// TwinCAT 3 PLC project TSG_swash_Neusiedl
// ProgramVersion: 3.1.4023.0
// libraries:
//   EfficientIO Communicator, * (EfficientIO)
//   Lynus Energy Basic, * (Lynus AG)
//   Lynus Energy ModbusTCP, * (Lynus AG)
//   Lynus Persistent Data V1, * (Lynus AG)
//   Lynus Standards, * (Lynus AG)
//   Tc2_MBus, * (Beckhoff Automation GmbH)
//   Tc2_ModbusSrv, * (Beckhoff Automation GmbH)
//   Tc2_Standard, * (Beckhoff Automation GmbH)
//   Tc2_System, * (Beckhoff Automation GmbH)
//   Tc2_Utilities, * (Beckhoff Automation GmbH)
//   Tc3_Module, * (Beckhoff Automation GmbH)
// project tree:
//   / FastTasks.TcTTO, PlcTask.TcTTO, SlowTasks.TcTTO
//   FB/ FB_ModBus_100Registers_FC4.TcPOU, FB_ModBus_100Registers_FC3.TcPOU, F_DWORD_TO_FLOAT32.TcPOU
//   POUs/ prgComLynus.TcPOU, prgEM.TcPOU, prgModbus.TcPOU, prgPersistent.TcPOU (not stored), prgPV.TcPOU, prgRWLynus.TcPOU, prgVarLynus.TcPOU, prgWCounter.TcPOU, prgWCounter_old.TcPOU (excluded from build), prg_SystemTime.TcPOU (not stored)
// real-time tasks:
//   TASK PlcTask: cycle T#10ms, priority 20, ADS port 350
//   TASK SlowTasks: cycle T#20ms, priority 21, ADS port 351
//   TASK FastTasks: cycle T#5ms, priority 19, ADS port 352
// I/O:
//   DEVICE Device 1 (Beckhoff CCAT)
//   DEVICE Device 3 (CX-BK)
//     Box 1 (CX-BK)
// variable links:
//   TSG_swash_Neusiedl/TSG_swash_Neusiedl Instance <-> Device 3 (CX-BK)/Box 1 (CX-BK)
//     FastTasks Inputs/prgWCounter.stComIn/D <-> Term 2 (KL6781)/Channel 1/Data In 0
//     FastTasks Inputs/prgWCounter.stComIn/D @bit {8..168 step 8} <-> Term 2 (KL6781)/Channel 1/Data In {1..21}  (21 links)
//     FastTasks Inputs/prgWCounter.stComIn/Status <-> Term 2 (KL6781)/Channel 1/Status
//     FastTasks Outputs/prgWCounter.stComOut/Ctrl <-> Term 2 (KL6781)/Channel 1/Ctrl
//     FastTasks Outputs/prgWCounter.stComOut/D <-> Term 2 (KL6781)/Channel 1/Data Out 0
//     FastTasks Outputs/prgWCounter.stComOut/D @bit {8..168 step 8} <-> Term 2 (KL6781)/Channel 1/Data Out {1..21}  (21 links)
//     PlcTask Inputs/prgEM.fbEM1.fbKL3403.byStateCH1 <-> Term 3 (KL3403)/Channel 1/State
//     PlcTask Inputs/prgEM.fbEM1.fbKL3403.byStateCH2 <-> Term 3 (KL3403)/Channel 2/State
//     PlcTask Inputs/prgEM.fbEM1.fbKL3403.byStateCH3 <-> Term 3 (KL3403)/Channel 3/State
//     PlcTask Inputs/prgEM.fbEM1.fbKL3403.iDataInCH1 <-> Term 3 (KL3403)/Channel 1/Data In
//     PlcTask Inputs/prgEM.fbEM1.fbKL3403.iDataInCH2 <-> Term 3 (KL3403)/Channel 2/Data In
//     PlcTask Inputs/prgEM.fbEM1.fbKL3403.iDataInCH3 <-> Term 3 (KL3403)/Channel 3/Data In
//     PlcTask Inputs/prgEM.fbKBusState.uiKBusState_OUT <-> Inputs/State
//     PlcTask Outputs/prgEM.fbEM1.fbKL3403.byCntrCH1 <-> Term 3 (KL3403)/Channel 1/Ctrl
//     PlcTask Outputs/prgEM.fbEM1.fbKL3403.byCntrCH2 <-> Term 3 (KL3403)/Channel 2/Ctrl
//     PlcTask Outputs/prgEM.fbEM1.fbKL3403.byCntrCH3 <-> Term 3 (KL3403)/Channel 3/Ctrl

CONFIGURATION TSG_swash_Neusiedl
    RESOURCE PLC ON TwinCAT3
        TASK FastTasks(INTERVAL := T#5ms, PRIORITY := 19);
        TASK PlcTask(INTERVAL := T#10ms, PRIORITY := 20);
        TASK SlowTasks(INTERVAL := T#20ms, PRIORITY := 21);
        PROGRAM prgRWLynus WITH FastTasks : prgRWLynus;
        PROGRAM prgVarLynus WITH FastTasks : prgVarLynus;
        PROGRAM prgWCounter WITH FastTasks : prgWCounter;
        PROGRAM prgPV WITH PlcTask : prgPV;
        PROGRAM prgEM WITH PlcTask : prgEM;
        PROGRAM prgModbus WITH PlcTask : prgModbus;
        PROGRAM prgPersistent WITH PlcTask : prgPersistent;
        PROGRAM prgComLynus WITH SlowTasks : prgComLynus;
    END_RESOURCE
END_CONFIGURATION

// ---- POUs/prgRWLynus.TcPOU
PROGRAM prgRWLynus
VAR
	fbRW1		: FB_ReadWrite_V2;
END_VAR

fbRW1(eUploadType:= eSelectDataUploadType.e_Change_Intervall5min, bBusy=> , bError=> , udiErrorCodeOut=> , eErrorReadWrite_Out=> );

END_PROGRAM

// ---- POUs/prgVarLynus.TcPOU
PROGRAM prgVarLynus
VAR
	fbVar			: FB_VarInfo;
END_VAR

fbVar(
	bReadInfo:= , 
	eTMCFile:= eSelectTMCFile.eDontUseTMCFile, 
	eSavePositionTMCFile:= eSavePositionOnPLC.ePostionHardDisk, 
	udiCounterFoundVariables=> , 
	bError=> , 
	bBusy=> , 
	byProgress=> , 
	udiErrorCodeOut=> , 
	eErrorVarInfo_Out=> , 
	sVarWithError=> );

END_PROGRAM

// ---- POUs/prgWCounter.TcPOU
PROGRAM prgWCounter
VAR
	fbMBusKL6781 : FB_MBUSKL6781;
	stComIn    AT %I*	:	ST_KL6781inData22B;
	stComOut   AT %Q*	:	ST_KL6781outData22B;
	stCom				:	ST_MBUS_Communication;
	fb_Mbus_11				: 	FB_MBUS_General_Water;
	fb_Mbus_12				: 	FB_MBUS_General_Water;
	fb_Mbus_13				: 	FB_MBUS_General_Water;
	fb_Mbus_14				: 	FB_MBUS_General_Water;
	fb_Mbus_15				: 	FB_MBUS_General_Water;
	fb_Mbus_16				: 	FB_MBUS_General_Water;
	fb_Mbus_17				: 	FB_MBUS_General_Water;
	fbmbusScan	: FB_MBUS_Scan;
	m_StartScan: BOOL;
	FB_ChangeAdress : FB_MBUS_ChangeAdr;
	lr_Water_Zisterne_Entnahme					: LREAL;						//{#lynus.ag#()}
	lr_Water_Frisch_Noteinspeisung				: LREAL;						//{#lynus.ag#()}
	lr_Water_Frischwasser_SB					: LREAL;						//{#lynus.ag#()}
	lr_Water_Innenreinigung						: LREAL;						//{#lynus.ag#()}
	lr_Water_Frisch_Absperrung_PO				: LREAL;						//{#lynus.ag#()}
	lr_Water_Absperrung_Zisterne				: LREAL;						//{#lynus.ag#()}
	lr_Water_FW_Zulauf_Zisterne					: LREAL;						//{#lynus.ag#()}
			
	m_Done			: BOOL;
	
END_VAR
VAR PERSISTENT
	lr_Water_Zisterne_Entnahme_LD				: LREAL;						//{#lynus.ag#()}
	lr_Water_Frisch_Noteinspeisung_LD			: LREAL;						//{#lynus.ag#()}
	lr_Water_Frischwasser_SB_LD					: LREAL;						//{#lynus.ag#()}
	lr_Water_Innenreinigung_LD					: LREAL;						//{#lynus.ag#()}
	lr_Water_Frisch_Absperrung_PO_LD			: LREAL;						//{#lynus.ag#()}
	lr_Water_Absperrung_Zisterne_LD				: LREAL;						//{#lynus.ag#()}
	lr_Water_FW_Zulauf_Zisterne_LD				: LREAL;						//{#lynus.ag#()}
	
	lr_Water_Zisterne_Entnahme_Old			: LREAL;						
	lr_Water_Frisch_Noteinspeisung_Old		: LREAL;						
	lr_Water_Frischwasser_SB_Old			: LREAL;						
	lr_Water_Innenreinigung_Old				: LREAL;						
	lr_Water_Frisch_Absperrung_PO_Old		: LREAL;						
	lr_Water_Absperrung_Zisterne_Old		: LREAL;						
	lr_Water_FW_Zulauf_Zisterne_Old			: LREAL;	
END_VAR



	
		

	
fbMBusKL6781(
	usiRetries:= , 
	bStart:= , 
	bDisabled:= , 
	bBusy=> , 
	bReady=> , 
	bError=> , 
	eError=> , 
	stComIn:= stComIn, 
	stComOut:= stComOut, 
	stCom:= stCom);

fb_Mbus_11(
	usiAddress:= 11 , 
	stSecAdr:= , 
	eBaudrate:= E_MBUS_Baudrate.eMBus_Baud2400, 
	bStart:= TRUE, 
	bSND_NKE:= , 
	bReadInit:= , 
	tMinSendTime:= T#10S , 
	bDisabled:= , 
	bBusy=> , 
	bReady=> , 
	bError=> , 
	eError=> , 
	dwIdNumber=> , 
	byStatus=> , 
	byGEN=> , 
	byCounter=> , 
	usiRecivedAdr=> , 
	eMedium=> , 
	sMan=> , 
	stVolume=> , 
	stFlow=> , 
	stCom:= stCom);
	
fb_Mbus_12(
	usiAddress:= 12 , 
	stSecAdr:= , 
	eBaudrate:= E_MBUS_Baudrate.eMBus_Baud2400, 
	bStart:= TRUE, 
	bSND_NKE:= , 
	bReadInit:= , 
	tMinSendTime:= T#10S , 
	bDisabled:= , 
	bBusy=> , 
	bReady=> , 
	bError=> , 
	eError=> , 
	dwIdNumber=> , 
	byStatus=> , 
	byGEN=> , 
	byCounter=> , 
	usiRecivedAdr=> , 
	eMedium=> , 
	sMan=> , 
	stVolume=> , 
	stFlow=> , 
	stCom:= stCom);
	
fb_Mbus_13(
	usiAddress:= 13 , 
	stSecAdr:= , 
	eBaudrate:= E_MBUS_Baudrate.eMBus_Baud2400, 
	bStart:= TRUE, 
	bSND_NKE:= , 
	bReadInit:= , 
	tMinSendTime:= T#10S , 
	bDisabled:= , 
	bBusy=> , 
	bReady=> , 
	bError=> , 
	eError=> , 
	dwIdNumber=> , 
	byStatus=> , 
	byGEN=> , 
	byCounter=> , 
	usiRecivedAdr=> , 
	eMedium=> , 
	sMan=> , 
	stVolume=> , 
	stFlow=> , 
	stCom:= stCom);	
	
fb_Mbus_14(
	usiAddress:= 14 , 
	stSecAdr:= , 
	eBaudrate:= E_MBUS_Baudrate.eMBus_Baud2400, 
	bStart:= TRUE, 
	bSND_NKE:= , 
	bReadInit:= , 
	tMinSendTime:= T#10S , 
	bDisabled:= , 
	bBusy=> , 
	bReady=> , 
	bError=> , 
	eError=> , 
	dwIdNumber=> , 
	byStatus=> , 
	byGEN=> , 
	byCounter=> , 
	usiRecivedAdr=> , 
	eMedium=> , 
	sMan=> , 
	stVolume=> , 
	stFlow=> , 
	stCom:= stCom);
	
fb_Mbus_15(
	usiAddress:= 15 , 
	stSecAdr:= , 
	eBaudrate:= E_MBUS_Baudrate.eMBus_Baud2400, 
	bStart:= TRUE, 
	bSND_NKE:= , 
	bReadInit:= , 
	tMinSendTime:= T#10S , 
	bDisabled:= , 
	bBusy=> , 
	bReady=> , 
	bError=> , 
	eError=> , 
	dwIdNumber=> , 
	byStatus=> , 
	byGEN=> , 
	byCounter=> , 
	usiRecivedAdr=> , 
	eMedium=> , 
	sMan=> , 
	stVolume=> , 
	stFlow=> , 
	stCom:= stCom);

fb_Mbus_16(
	usiAddress:= 16 , 
	stSecAdr:= , 
	eBaudrate:= E_MBUS_Baudrate.eMBus_Baud2400, 
	bStart:= TRUE, 
	bSND_NKE:= , 
	bReadInit:= , 
	tMinSendTime:= T#10S , 
	bDisabled:= , 
	bBusy=> , 
	bReady=> , 
	bError=> , 
	eError=> , 
	dwIdNumber=> , 
	byStatus=> , 
	byGEN=> , 
	byCounter=> , 
	usiRecivedAdr=> , 
	eMedium=> , 
	sMan=> , 
	stVolume=> , 
	stFlow=> , 
	stCom:= stCom);

fb_Mbus_17(
	usiAddress:= 17 , 
	stSecAdr:= , 
	eBaudrate:= E_MBUS_Baudrate.eMBus_Baud2400, 
	bStart:= TRUE, 
	bSND_NKE:= , 
	bReadInit:= , 
	tMinSendTime:= T#10S , 
	bDisabled:= , 
	bBusy=> , 
	bReady=> , 
	bError=> , 
	eError=> , 
	dwIdNumber=> , 
	byStatus=> , 
	byGEN=> , 
	byCounter=> , 
	usiRecivedAdr=> , 
	eMedium=> , 
	sMan=> , 
	stVolume=> , 
	stFlow=> , 
	stCom:= stCom);


lr_Water_Frisch_Noteinspeisung	 			:= UDINT_TO_LREAL(LREAL_TO_UDINT((STRING_TO_LREAL(fb_Mbus_11.stVolume.sValue)*1000)))/1000;
lr_Water_Frischwasser_SB	 				:= UDINT_TO_LREAL(LREAL_TO_UDINT((STRING_TO_LREAL(fb_Mbus_12.stVolume.sValue)*1000)))/1000;
lr_Water_Innenreinigung						:= UDINT_TO_LREAL(LREAL_TO_UDINT((STRING_TO_LREAL(fb_Mbus_13.stVolume.sValue)*1000)))/1000;
lr_Water_Frisch_Absperrung_PO		 		:= UDINT_TO_LREAL(LREAL_TO_UDINT((STRING_TO_LREAL(fb_Mbus_14.stVolume.sValue)*1000)))/1000;
lr_Water_Zisterne_Entnahme	 				:= UDINT_TO_LREAL(LREAL_TO_UDINT((STRING_TO_LREAL(fb_Mbus_15.stVolume.sValue)*1000)))/1000;
lr_Water_Absperrung_Zisterne				:= UDINT_TO_LREAL(LREAL_TO_UDINT((STRING_TO_LREAL(fb_Mbus_16.stVolume.sValue)*1000)))/1000;
lr_Water_FW_Zulauf_Zisterne		 			:= UDINT_TO_LREAL(LREAL_TO_UDINT((STRING_TO_LREAL(fb_Mbus_17.stVolume.sValue)*1000)))/1000;


	
(* only required for commissioning the water meters	
fbMBusScan(		bStart:= m_StartScan, 
				bStop:= NOT m_StartScan, 
				eBaudrate:= E_MBUS_Baudrate.eMBus_Baud2400, 
				bDisabled:= , 
				bBusy=> , 
				bReady=> , 
				bError=> , 
				eError=> , 
				usiAddress=> , 
				usiCount=> , 
				arrDevice=> , 
				stCom:= stCom);

FB_ChangeAdress(	usiAdrOld:= usi_Old, 
					usiAdrNew:= usi_New, 
					eBaudrate:= E_MBUS_Baudrate.eMBus_Baud2400, 
					bStart:= m_Start_Change, 
					bDisabled:= m_Disable_Change, 
					bBusy=> , 
					bReady=> , 
					bError=> , 
					eError=> , 
					stCom:= stCom);
*)

// save every day at 23:59 the water counter and calculate the consumption of the last 24h


// store water counters and calculate the consumtion of the last day

prg_SystemTime ();
IF prg_SystemTime.structSystemTime.wHour =23 AND prg_SystemTime.structSystemTime.wMinute=59 AND prg_SystemTime.structSystemTime.wSecond = 59 AND NOT m_Done THEN
	
	lr_Water_Zisterne_Entnahme_LD 		:= lr_Water_Zisterne_Entnahme - lr_Water_Zisterne_Entnahme_Old;
	lr_Water_Frisch_Noteinspeisung_LD	:= lr_Water_Frisch_Noteinspeisung - lr_Water_Frisch_Noteinspeisung_Old;
	lr_Water_Frischwasser_SB_LD			:= lr_Water_Frischwasser_SB - lr_Water_Frischwasser_SB_old;							
	lr_Water_Innenreinigung_LD			:= lr_Water_Innenreinigung - lr_Water_Innenreinigung_Old;										
	lr_Water_Frisch_Absperrung_PO_LD	:= lr_Water_Frisch_Absperrung_PO - lr_Water_Frisch_Absperrung_PO_Old;
	lr_Water_Absperrung_Zisterne_LD  	:= lr_Water_Absperrung_Zisterne - lr_Water_Absperrung_Zisterne_old;
	lr_Water_FW_Zulauf_Zisterne_LD		:= lr_Water_FW_Zulauf_Zisterne - lr_Water_FW_Zulauf_Zisterne_Old;
	
		
	lr_Water_Zisterne_Entnahme_Old 		:= lr_Water_Zisterne_Entnahme;	
	lr_Water_Frisch_Noteinspeisung_Old	:= lr_Water_Frisch_Noteinspeisung	;					
	lr_Water_Frischwasser_SB_Old		:= lr_Water_Frischwasser_SB		;		
	lr_Water_Innenreinigung_Old			:= lr_Water_Innenreinigung			;					
	lr_Water_Frisch_Absperrung_PO_Old	:= lr_Water_Frisch_Absperrung_PO	;				
	lr_Water_Absperrung_Zisterne_Old	:= lr_Water_Absperrung_Zisterne	;		
	lr_Water_FW_Zulauf_Zisterne_Old		:= lr_Water_FW_Zulauf_Zisterne		;
	m_Done := TRUE;
END_IF

IF prg_SystemTime.structSystemTime.wHour =0 AND prg_SystemTime.structSystemTime.wMinute=0 then 
 	m_Done := FALSE;
END_IF

END_PROGRAM

// ---- POUs/prgPV.TcPOU
PROGRAM prgPV
VAR
	fbPV					: FB_Symo_PV_Inverter_FLOAT_1_DM_1_Inverter;
	fbPVInt					: FB_PV_Power;
	fbPVCounter				: FB_EnergyCounter;
	lrPowerPV				: LREAL;				//{#lynus.ag#()}
	byErrorWarningPV		: BYTE;					//{#lynus.ag#()}
	bReadyPD_PV				: BOOL;					//{#lynus.ag#()}
	byErrorWarningPD_PV		: BYTE;					//{#lynus.ag#()}
	rHeartbeat_PD_PV		: REAL;					//{#lynus.ag#()}
END_VAR
VAR PERSISTENT
	lrCounterPV				: LREAL;				//{#lynus.ag#()}
END_VAR

fbPV(
	bEnable:= TRUE, 
	sIPAdress:= '192.168.71.73', 
	byUnitID_Inverter:= 1, 
	stDataSymo10=> , 
	stDataEMPower_PV=> , 
	stDataEMCounter_PV=> , 
	diNrOfEM_OUT_PV=> );
	
fbPVInt(
	bEnable:= TRUE, 
	bPowerDataInvers:= , 
	diNrOfEM_IN_PV:= fbPV.diNrOfEM_OUT_PV, 
	stDataPv=> , 
	diNrOfPv_OUT=> );
	
lrPowerPV := fbPVInt.stDataPv.lrPower;
	byErrorWarningPV := fbPVInt.stDataPv.byErrorWarning;
	

// EnergyCounter
fbPVCounter(
	byActiveTariff:= 1, 
	lrPowerInput:= 0 - lrPowerPV, 
	lrTotalCounterEnergy_Consumption=> , 
	lrTotalCounterEnergy_Production=> , 
	lrCounterEnergyT1_Consumption=> , 
	lrCounterEnergyT2_Consumption=> , 
	lrCounterEnergyT1_Production=> , 
	lrCounterEnergyT2_Production=> );
	
IF fbPVCounter.lrTotalCounterEnergy_Production > lrCounterPV THEN  	
	lrCounterPV := fbPVCounter.lrTotalCounterEnergy_Production;
END_IF

END_PROGRAM

// ---- POUs/prgEM.TcPOU
PROGRAM prgEM
VAR
	fbKBusState		: FB_K_Bus_State;
	fbEM1			: FB_EM_Beckhoff_KL3403;
	bGridEnabled	: BOOL;								//{#lynus.ag#()}
	lrPowerGrid		: LREAL;							//{#lynus.ag#()}
	lrPowerEM1_1	: LREAL;							//{#lynus.ag#()}
	lrPowerEM1_2	: LREAL;							//{#lynus.ag#()}
	lrPowerEM1_3	: LREAL;							//{#lynus.ag#()}
	lrCounterGrid	: LREAL;							//{#lynus.ag#()}
	lrApparentPowerEM: LREAL;						//{#lynus.ag#()}
	lrReactivePowerEM: LREAL;						//{#lynus.ag#()}
END_VAR
VAR PERSISTENT
	bEnableGrid		: BOOL;							//{#lynus.ag#()}
END_VAR

//The mapping of this function must be linked with the K-Bus State in the E/A Part
fbKBusState(uiKBusState_OUT=> );

//The mapping of this function must be linked with the KL3403 in the E/A Part
fbEM1(
	bEnable:= bEnableGrid, 
	bChannel1Invers:= FALSE,				//Invert power data when transformer are mounted upside down
	bChannel2Invers:= FALSE,
	bChannel3Invers:= FALSE,
	uiCurrentTransformerRatioL1:= 400, //Transformer ratio on the secondary side
	uiCurrentTransformerRatioL2:= 400, 
	uiCurrentTransformerRatioL3:= 400, 
	uiKBusState_IN:= fbKBusState.uiKBusState_OUT, 
	stDataEMPower=> , 
	stDataEMCounter=> , 
	stDataEMPowerRealTime=> , 
	stDataEMCounterRealTime=> , 
	diNrOfEM_OUT=> );

lrPowerGrid := fbEM1.stDataEMPower.lrPowerTotal;
lrCounterGrid := fbEM1.stDataEMCounter.lrTotalCounterEnergy_Consumption;	
lrPowerEM1_1 := fbEM1.stDataEMPower.lrPowerL1;
lrPowerEM1_2 := fbEM1.stDataEMPower.lrPowerL2;
lrPowerEM1_3 := fbEM1.stDataEMPower.lrPowerL3;
bGridEnabled := fbEM1.bEnable;
lrApparentPowerEM := fbEM1.stDataEMPower.lrApparentPowerTotal;
lrReactivePowerEM := fbEM1.stDataEMPower.lrReactivePowerTotal;

END_PROGRAM

// ---- POUs/prgModbus.TcPOU
PROGRAM prgModbus
VAR
	FB_Modbus: FB_ModBus_100Registers_FC4;
	FB_Modbus1: FB_ModBus_100Registers_FC3;
	m_Enable: BOOL:=TRUE;
	m_Enable1: BOOL:=TRUE;
	fbConvertWordToDword		: FB_CV_WORD_TO_DWORD;			//Convert Word to Dword
	usintSign					: USINT;						// converstion dword to real	
	intExponent					: INT;							// converstion dword to real
	realMantisse				: REAL;							// converstion dword to real
	x: INT;
	r_HP_OutsideTemp	: REAL;									//{#lynus.ag#()}
	r_HP_SupplyTemp		: REAL;									//{#lynus.ag#()}
	r_HP_ReturnTemp		: REAL;									//{#lynus.ag#()}
	r_HP_SupplyTemp_A	: REAL;									//{#lynus.ag#()}
	r_HP_SupplyTemp_B	: REAL;									//{#lynus.ag#()}
	r_HP_SupplyTemp_C	: REAL;									//{#lynus.ag#()}
	r_HP_Heissgastemperatur: REAL;								//{#lynus.ag#()}
	r_HP_AirSupplyTemp: REAL;									//{#lynus.ag#()}
	r_HP_AirHeatExchangerTemp: REAL;							//{#lynus.ag#()}
	r_HP_AverageOutsideTemp: REAL;								//{#lynus.ag#()}
	r_HP_HeatQuantitySupply: REAL;								//{#lynus.ag#()}
	m_HP_SystemMode_Off: BOOL;									//{#lynus.ag#()}
	m_HP_SystemMode_Auto: BOOL;									//{#lynus.ag#()}
	m_HP_SystemMode_OnlyWater: BOOL;							//{#lynus.ag#()}
	m_HP_SystemMode_OnceCharging: BOOL;							//{#lynus.ag#()}
	m_HP_HeatingMode_Off: BOOL;									//{#lynus.ag#()}
	m_HP_HeatingMode_Time: BOOL;								//{#lynus.ag#()}
	m_HP_HeatingMode_Normal: BOOL;								//{#lynus.ag#()}
	m_HP_HeatingMode_ECO: BOOL;									//{#lynus.ag#()}
	m_HP_HeatingMode_Manual: BOOL;								//{#lynus.ag#()}
END_VAR

FB_Modbus(
	m_Enable:=m_Enable , 
	str_IPAdress:='192.168.71.71' , 
	w_Adress:= 1000, 
	usint_Quantity:= 70, 
	m_PollSuccessful=> , 
	w_Array_Received=> , 
	udint_Error_ID=> );
	
FB_Modbus1(
	m_Enable:=m_Enable1 , 
	str_IPAdress:='192.168.71.71' , 
	w_Adress:= 2000, 
	usint_Quantity:= 4, 
	m_PollSuccessful=> , 
	w_Array_Received=> , 
	udint_Error_ID=> );

x:=1; 	//1000	Außentemperatur
r_HP_OutsideTemp  			:= F_DWORD_TO_FLOAT32(dwInput := WORD_TO_DWORD(FB_Modbus.w_Array_Received[x]) + 16#10000 * WORD_TO_DWORD(FB_Modbus.w_Array_Received[x+1]));
x:=3;	//1002	Wärmepumpen Vorlauftemperatur
r_HP_SupplyTemp  			:= F_DWORD_TO_FLOAT32(dwInput := WORD_TO_DWORD(FB_Modbus.w_Array_Received[x]) + 16#10000 * WORD_TO_DWORD(FB_Modbus.w_Array_Received[x+1]));
x:=9;	//1008	Wärmepumpen Rücklauftemperatur / Wärmespeichertemperatur
r_HP_ReturnTemp  			:= F_DWORD_TO_FLOAT32(dwInput := WORD_TO_DWORD(FB_Modbus.w_Array_Received[x]) + 16#10000 * WORD_TO_DWORD(FB_Modbus.w_Array_Received[x+1]));
x:=17;	//1016	Heizkreis A Vorlauftemperatur
r_HP_SupplyTemp_A  			:= F_DWORD_TO_FLOAT32(dwInput := WORD_TO_DWORD(FB_Modbus.w_Array_Received[x]) + 16#10000 * WORD_TO_DWORD(FB_Modbus.w_Array_Received[x+1]));
x:=19;	//1018	Heizkreis B Vorlauftemperatur
r_HP_SupplyTemp_B  			:= F_DWORD_TO_FLOAT32(dwInput := WORD_TO_DWORD(FB_Modbus.w_Array_Received[x]) + 16#10000 * WORD_TO_DWORD(FB_Modbus.w_Array_Received[x+1]));
x:=21;	//1020	Heizkreis C Vorlauftemperatur
r_HP_SupplyTemp_C  			:= F_DWORD_TO_FLOAT32(dwInput := WORD_TO_DWORD(FB_Modbus.w_Array_Received[x]) + 16#10000 * WORD_TO_DWORD(FB_Modbus.w_Array_Received[x+1]));
x:=45;	//1044	Heissgastemperatur
r_HP_Heissgastemperatur  	:= F_DWORD_TO_FLOAT32(dwInput := WORD_TO_DWORD(FB_Modbus.w_Array_Received[x]) + 16#10000 * WORD_TO_DWORD(FB_Modbus.w_Array_Received[x+1]));
x:=49;	//1044	Heissgastemperatur
r_HP_AirSupplyTemp 			:= F_DWORD_TO_FLOAT32(dwInput := WORD_TO_DWORD(FB_Modbus.w_Array_Received[x]) + 16#10000 * WORD_TO_DWORD(FB_Modbus.w_Array_Received[x+1]));
x:=51;	//1050	Luftwärmetauschertemperatur
r_HP_AirHeatExchangerTemp 	:= F_DWORD_TO_FLOAT32(dwInput := WORD_TO_DWORD(FB_Modbus.w_Array_Received[x]) + 16#10000 * WORD_TO_DWORD(FB_Modbus.w_Array_Received[x+1])); 
x:=61;	//1060	Gemittelte Aussentemperatur
r_HP_AverageOutsideTemp 	:= F_DWORD_TO_FLOAT32(dwInput := WORD_TO_DWORD(FB_Modbus.w_Array_Received[x]) + 16#10000 * WORD_TO_DWORD(FB_Modbus.w_Array_Received[x+1]));
x:=69;	//1068	Wärmemenge Wärmepumpenvorlauf
r_HP_HeatQuantitySupply		:= F_DWORD_TO_FLOAT32(dwInput := WORD_TO_DWORD(FB_Modbus.w_Array_Received[x]) + 16#10000 * WORD_TO_DWORD(FB_Modbus.w_Array_Received[x+1]));


//2000	Betriebsart System
CASE FB_Modbus1.w_Array_Received[1] OF
	0:
	m_HP_SystemMode_Off				:= TRUE;
	m_HP_SystemMode_Auto			:= FALSE;
	m_HP_SystemMode_OnlyWater		:= FALSE;
	m_HP_SystemMode_OnceCharging	:= FALSE;
	1:
	m_HP_SystemMode_Off				:= FALSE;
	m_HP_SystemMode_Auto			:= TRUE;
	m_HP_SystemMode_OnlyWater		:= FALSE;
	m_HP_SystemMode_OnceCharging	:= FALSE;
	2:
	m_HP_SystemMode_Off				:= FALSE;
	m_HP_SystemMode_Auto			:= FALSE;
	m_HP_SystemMode_OnlyWater		:= TRUE;
	m_HP_SystemMode_OnceCharging	:= FALSE;
	3:
	m_HP_SystemMode_Off				:= FALSE;
	m_HP_SystemMode_Auto			:= FALSE;
	m_HP_SystemMode_OnlyWater		:= FALSE;
	m_HP_SystemMode_OnceCharging	:= TRUE;
END_CASE


//2002	Betriebsart Heizkreis
CASE FB_Modbus1.w_Array_Received[1] OF
	0:
	m_HP_HeatingMode_Off			:= TRUE;
	m_HP_HeatingMode_Time			:= FALSE;
	m_HP_HeatingMode_Normal			:= FALSE;
	m_HP_HeatingMode_ECO			:= FALSE;
	m_HP_HeatingMode_Manual			:= FALSE;
	1:
	m_HP_HeatingMode_Off			:= FALSE;
	m_HP_HeatingMode_Time			:= TRUE;
	m_HP_HeatingMode_Normal			:= FALSE;
	m_HP_HeatingMode_ECO			:= FALSE;
	m_HP_HeatingMode_Manual			:= FALSE;
	2:
	m_HP_HeatingMode_Off			:= FALSE;
	m_HP_HeatingMode_Time			:= FALSE;
	m_HP_HeatingMode_Normal			:= TRUE;
	m_HP_HeatingMode_ECO			:= FALSE;
	m_HP_HeatingMode_Manual			:= FALSE;
	3:
	m_HP_HeatingMode_Off			:= FALSE;
	m_HP_HeatingMode_Time			:= FALSE;
	m_HP_HeatingMode_Normal			:= FALSE;
	m_HP_HeatingMode_ECO			:= TRUE;
	m_HP_HeatingMode_Manual			:= FALSE;
	4:
	m_HP_HeatingMode_Off			:= FALSE;
	m_HP_HeatingMode_Time			:= FALSE;
	m_HP_HeatingMode_Normal			:= FALSE;
	m_HP_HeatingMode_ECO			:= FALSE;
	m_HP_HeatingMode_Manual			:= TRUE;
END_CASE

END_PROGRAM

// ---- FB/FB_ModBus_100Registers_FC4.TcPOU
FUNCTION_BLOCK FB_ModBus_100Registers_FC4
VAR_INPUT PERSISTENT
	m_Enable					: BOOL;						//Enable the Fuctionblock and his logic
	str_IPAdress				: STRING(15);				//IP Adress of the meter
	w_Adress					: WORD;						//modbus adress
	usint_Quantity				: USINT;						//Number of Words to get polled, max 100
END_VAR
VAR_OUTPUT
	m_PollSuccessful			: BOOL;						//Poll succesfull		
	w_Array_Received			: ARRAY[1..100] OF WORD;	// received data
	udint_Error_ID				: UDINT;					// ERR ID FB_MBReadRegs
END_VAR
VAR
	{attribute 'hide'}
	timer_Delay					: TON;						//Timer for Delay between Requests
	{attribute 'hide'}
	timer_DelayStart			: TON;						//Timer to start the state machine with Delay after enabling or after the system ist restartet
	{attribute 'hide'}
	timer_TimeOut				: TON;						//Timer for Timeout MB Read
	{attribute 'hide'}
	iStateModbusRead			: INT;						//State machine for read out Data over Modbus RTU
	{attribute 'hide'}
	fbMBRead_FC4				: FB_MBReadInputRegs ;		//Modbus Read Function (FC4)
	{attribute 'hide'}
	ftrig_PEnable				: f_trig;					//Internal positive Edge
	{attribute 'hide'}
	iStateModbusError			: INT;						//State machine for error out Data over Modbus TCP/IP	
	{attribute 'hide'}
	FPError_FC_4				: R_TRIG;					//Internal positive Edge
	{attribute 'hide'}
	arrBuffer_FC4				: ARRAY[1..100] OF WORD;		//Buffer with Data from FC3
	{attribute 'hide'}
	timer_Connection_ok			: TON;
	int_Data_Received			: INT;
	{attribute 'hide'}
	m_MBTCPError				: BOOL;
	{attribute 'hide'}
	int_Data_Received_old		: INT;
	{attribute 'hide'}
	timer_Connection_ok_TOF	: TOF;
	{attribute 'hide'}
	fbConvertWordToDword		: FB_CV_WORD_TO_DWORD;			//Convert Word to Dword
	{attribute 'hide'}
	m_Poll_ok: BOOL;
	{attribute 'hide'}
	timer_Wait: Ton;
	int_TimeoutError: INT;
	int_FC3Error: INT;
END_VAR

(*--------------------------------------------------------------------------------------------Limits-------------------------------------------------------------------------------------*)

w_Adress := LIMIT(0,w_Adress,32767);
usint_Quantity := LIMIT(1,usint_Quantity,100);
	
(*--------------------------------------------------------------------------------------------State Machine Read--------------------------------------------------------------------------------------*)

//Timer for Delay
timer_Delay(IN:= , PT:= T#50MS, Q=> , ET=> );

//Timeout Timer is dissabled when the Init Step is aktiv or the function is not enabled
IF iStateModbusRead = 0 OR NOT m_Enable THEN 
	timer_Timeout.IN := FALSE; 
END_IF
timer_Timeout(IN:= , PT:= T#1S, Q=> , ET=> );

//Enable with Delay that not all sockets have to be created at the same time
timer_DelayStart(IN:= m_Enable, PT:= T#1S, Q=> , ET=> );
ftrig_PEnable(CLK:= timer_DelayStart.Q, Q=> );

IF ftrig_PEnable.Q AND iStateModbusRead = 0 THEN 
	iStateModbusRead := 1; 
END_IF		
		
//Not Enabled
IF NOT m_Enable THEN 
	iStateModbusRead := 0; 
	iStateModbusError := 0; 
END_IF		
		
CASE iStateModbusRead OF

	0://Init Step 
		timer_Delay.IN := FALSE;
		fbMBRead_FC4.bExecute := FALSE;
		m_Poll_ok:=FALSE;
		int_Data_Received:=0;
	
		iStateModbusRead := 1;
	
	1://read the required registers
		//Start Read
		fbMBRead_FC4.nQuantity := usint_Quantity;
		fbMBRead_FC4.nMBAddr := w_Adress;
		fbMBRead_FC4.bExecute := TRUE;
		fbMBRead_FC4.nUnitID := 1;
		timer_Timeout.IN := TRUE;
		IF fbMBRead_FC4.bBusy THEN 
			timer_Delay.IN := TRUE; 
		END_IF
		
		//Wait for Delay, copy Data and then next step
		IF NOT fbMBRead_FC4.bBusy AND NOT fbMBRead_FC4.bError AND timer_Delay.Q THEN
			m_Poll_ok:=TRUE;
			int_Data_Received:=int_Data_Received+1;
			m_MBTCPError := FALSE; 
			
			w_Array_Received := arrBuffer_FC4;
			
			
			//Go to Next Step
			timer_Timeout.IN := FALSE;
			fbMBRead_FC4.bExecute := FALSE;
			timer_Delay.IN := FALSE;		
			iStateModbusRead := 3;
		END_IF	

		//Error or Timeout
		IF FPError_FC_4.Q THEN 
			iStateModbusError := 300;
			int_FC3Error := int_FC3Error+1;
		ELSIF timer_Timeout.Q THEN   
			timer_Timeout.IN := FALSE;	
			iStateModbusError := 300;
			int_TimeoutError := int_TimeoutError+1;
		END_IF
		
	
	3://Wait and go to step 1
		//1 because 0 is the Init Step for Read
		timer_Wait.IN := TRUE;
		
		IF timer_Wait.Q = TRUE THEN
			iStateModbusRead := 1;
			timer_Wait.IN :=FALSE;
		END_IF

			
		
		//Error on Master, changes on Inputs or Timeout
		IF timer_Timeout.Q THEN 
			iStateModbusError := 300; 
		END_IF
	
END_CASE

(* wait timer*)

timer_Wait(PT:=T#3S);


(*------------------------------------------------------------------Error and Warning----------------------------------------------------------------------------*)	
 
timer_Connection_ok			(In:=int_Data_Received<>int_Data_Received_old,PT:=T#10S);
timer_Connection_ok_TOF		(In:=NOT(int_Data_Received<>int_Data_Received_old) AND int_Data_Received>3 ,PT:=T#20S);
int_Data_Received_old:=int_Data_Received;
m_PollSuccessful:=NOT timer_Connection_ok.Q AND timer_Connection_ok_TOF.Q ;

(*------------------------------------------------------------------------------------------Modbus TCP Functions---------------------------------------------------------------------------------------------*)

fbMBRead_FC4(	sIPAddr:= str_IPAdress, 
				nTCPPort:= 502,
				cbLength:= SIZEOF(arrBuffer_FC4), 
				pDestAddr:= ADR(arrBuffer_FC4), 
				tTimeout:= T#10S,
				nErrId => udint_Error_ID);

FPError_FC_4(CLK:= fbMBRead_FC4.  bError, Q=> );		

(*------------------------------------------------------------------------------------------State Machine Error---------------------------------------------------------------------------------------------*)	

CASE iStateModbusError OF
	
	300://Error
		timer_Wait.IN :=TRUE;
		timer_Delay.IN := FALSE;
		fbMBRead_FC4.bExecute := FALSE;
		m_MBTCPError := TRUE; 		
		m_Poll_ok:=FALSE;
		int_Data_Received:=0;
				//Restart from new with the Read out part after an Error
		IF timer_Wait.Q = TRUE THEN
			iStateModbusRead := 0;	
			iStateModbusError := 0;
			timer_Wait.IN :=FALSE;
			timer_Timeout.IN := FALSE;
		END_IF		
							
END_CASE

END_FUNCTION_BLOCK

// ---- FB/FB_ModBus_100Registers_FC3.TcPOU
FUNCTION_BLOCK FB_ModBus_100Registers_FC3
VAR_INPUT PERSISTENT
	m_Enable					: BOOL;						//Enable the Fuctionblock and his logic
	str_IPAdress				: STRING(15);				//IP Adress of the meter
	w_Adress					: WORD;						//modbus adress
	usint_Quantity				: usINT;						//Number of Words to get polled, max 100
END_VAR
VAR_OUTPUT
	m_PollSuccessful			: BOOL;						//Poll succesfull		
	w_Array_Received			: ARRAY[1..100] OF WORD;	// received data
	udint_Error_ID				: UDINT;					// ERR ID FB_MBReadRegs
END_VAR
VAR
	
	timer_Delay					: TON;						//Timer for Delay between Requests
	
	timer_DelayStart			: TON;						//Timer to start the state machine with Delay after enabling or after the system ist restartet
	
	timer_TimeOut				: TON;						//Timer for Timeout MB Read
	
	iStateModbusRead			: INT;						//State machine for read out Data over Modbus RTU
	
	fbMBRead_FC3				: FB_MBReadRegs  ;		//Modbus Read Function (FC3)
	
	ftrig_PEnable				: f_trig;					//Internal positive Edge
	
	iStateModbusError			: INT;						//State machine for error out Data over Modbus TCP/IP	
	
	FPError_FC_3				: R_TRIG;					//Internal positive Edge
	
	arrBuffer_FC3				: ARRAY[1..100] OF WORD;		//Buffer with Data from FC3
	
	timer_Connection_ok			: TON;
	int_Data_Received			: INT;
	
	m_MBTCPError				: BOOL;
	
	int_Data_Received_old		: INT;
	
	timer_Connection_ok_TOF	: TOF;
	
	fbConvertWordToDword		: FB_CV_WORD_TO_DWORD;			//Convert Word to Dword
	
	m_Poll_ok: BOOL;
	
	timer_Wait: Ton;
	int_TimeoutError: INT;
	int_FC3Error: INT;

END_VAR

(*	{attribute 'hide'}--------------------------------------------------------------------------------------------Limits-------------------------------------------------------------------------------------*)

w_Adress := LIMIT(0,w_Adress,32767);
usint_Quantity := LIMIT(1,usint_Quantity,100);
	
(*--------------------------------------------------------------------------------------------State Machine Read--------------------------------------------------------------------------------------*)

//Timer for Delay
timer_Delay(IN:= , PT:= T#50MS, Q=> , ET=> );

//Timeout Timer is dissabled when the Init Step is aktiv or the function is not enabled
IF iStateModbusRead = 0 OR NOT m_Enable THEN 
	timer_Timeout.IN := FALSE; 
END_IF
timer_Timeout(IN:= , PT:= T#1S, Q=> , ET=> );

//Enable with Delay that not all sockets have to be created at the same time
timer_DelayStart(IN:= m_Enable, PT:= T#1S, Q=> , ET=> );
ftrig_PEnable(CLK:= timer_DelayStart.Q, Q=> );

IF ftrig_PEnable.Q AND iStateModbusRead = 0 THEN 
	iStateModbusRead := 1; 
END_IF		
		
//Not Enabled
IF NOT m_Enable THEN 
	iStateModbusRead := 0; 
	iStateModbusError := 0; 
END_IF		
		
CASE iStateModbusRead OF

	0://Init Step 
		timer_Delay.IN := FALSE;
		fbMBRead_FC3.bExecute := FALSE;
		m_Poll_ok:=FALSE;
		int_Data_Received:=0;
	
		iStateModbusRead := 1;
	
	1://read the required registers
		//Start Read
		fbMBRead_FC3.nQuantity := usint_Quantity;
		fbMBRead_FC3.nMBAddr := w_Adress;
		fbMBRead_FC3.bExecute := TRUE;
		fbMBRead_FC3.nUnitID := 1;
		timer_Timeout.IN := TRUE;
		IF fbMBRead_FC3.bBusy THEN 
			timer_Delay.IN := TRUE; 
		END_IF
		
		//Wait for Delay, copy Data and then next step
		IF NOT fbMBRead_FC3.bBusy AND NOT fbMBRead_FC3.bError AND timer_Delay.Q THEN
			m_Poll_ok:=TRUE;
			int_Data_Received:=int_Data_Received+1;
			m_MBTCPError := FALSE; 
			
			w_Array_Received := arrBuffer_FC3;
			
			
			//Go to Next Step
			timer_Timeout.IN := FALSE;
			fbMBRead_FC3.bExecute := FALSE;
			timer_Delay.IN := FALSE;		
			iStateModbusRead := 3;
		END_IF	

		//Error or Timeout
		IF FPError_FC_3.Q THEN 
			iStateModbusError := 300;
			int_FC3Error := int_FC3Error+1;
		ELSIF timer_Timeout.Q THEN  
			timer_Timeout.IN := FALSE; 	
			iStateModbusError := 300;
			int_TimeoutError := int_TimeoutError+1;
		END_IF
		
	
	3://Wait and go to step 1
		//1 because 0 is the Init Step for Read
		timer_Wait.IN := TRUE;
		
		IF timer_Wait.Q = TRUE THEN
			iStateModbusRead := 1;
			timer_Wait.IN :=FALSE;
		END_IF

			
		
		//Error on Master, changes on Inputs or Timeout
		IF timer_Timeout.Q THEN 
			iStateModbusError := 300; 
		END_IF
	
END_CASE

(* wait timer*)

timer_Wait(PT:=T#3S);


(*------------------------------------------------------------------Error and Warning----------------------------------------------------------------------------*)	
 
timer_Connection_ok			(In:=int_Data_Received<>int_Data_Received_old,PT:=T#10S);
timer_Connection_ok_TOF		(In:=NOT(int_Data_Received<>int_Data_Received_old) AND int_Data_Received>3 ,PT:=T#20S);
int_Data_Received_old:=int_Data_Received;
m_PollSuccessful:=NOT timer_Connection_ok.Q AND timer_Connection_ok_TOF.Q ;

(*------------------------------------------------------------------------------------------Modbus TCP Functions---------------------------------------------------------------------------------------------*)

fbMBRead_FC3(	sIPAddr:= str_IPAdress, 
				nTCPPort:= 502,
				cbLength:= SIZEOF(arrBuffer_FC3), 
				pDestAddr:= ADR(arrBuffer_FC3), 
				tTimeout:= T#10S,
				nErrId => udint_Error_ID);

FPError_FC_3(CLK:= fbMBRead_FC3.bError, Q=> );		

(*------------------------------------------------------------------------------------------State Machine Error---------------------------------------------------------------------------------------------*)	

CASE iStateModbusError OF
	
	300://Error
		timer_Wait.IN :=TRUE;
		timer_Delay.IN := FALSE;
		fbMBRead_FC3.bExecute := FALSE;
		m_MBTCPError := TRUE; 		
		m_Poll_ok:=FALSE;
		int_Data_Received:=0;
				//Restart from new with the Read out part after an Error
		IF timer_Wait.Q = TRUE THEN
			iStateModbusRead := 0;	
			iStateModbusError := 0;
			timer_Wait.IN :=FALSE;
			timer_Timeout.IN := FALSE;
		END_IF		
							
END_CASE

END_FUNCTION_BLOCK

// ---- FB/F_DWORD_TO_FLOAT32.TcPOU
FUNCTION F_DWORD_TO_FLOAT32 : REAL
VAR_INPUT
	dwInput: DWORD;
END_VAR
VAR
	realSign: REAL;
	realExponent: REAL;
	realMantisse: REAL;
END_VAR

(* Sign *)
realSign:=BOOL_TO_REAL(dwInput.31);

(* Exponent *)
realExponent:=SHR(dwInput,23) AND 16#FF;

(* Mantisse *)
realMantisse:=dwInput AND 16#7FFFFF;

(* Result *)
F_DWORD_TO_FLOAT32:=EXPT((-1),realSign)*(1+realMantisse/8388608)*EXPT(2,realExponent-127);

END_FUNCTION

// ---- POUs/prgComLynus.TcPOU
PROGRAM prgComLynus
VAR
	fbCom			: FB_MqttCommunicator_V2;
END_VAR

fbCom(
	bConnect:= TRUE, 
	strAuthKey:= 'TSG88376368072' , 
	sUserName:= 'a242cb33-7d00-431c-a780-261995d86f3c', 
	sUserPassword:= '68bc2b87-a9ad-4107-814c-33cbf7ba0678' , 
	eSavePositionCertificate:= eSavePositionOnPLC.ePostionHardDisk,  
	bConnected=> , 
	bError=> , 
	hrErrorCode=> , 
	eConnectionState=> , 
	eErrorMessage_Out=> );

(*
fbCom(
	bConnect:= TRUE, 
	sUserName:= 'a242cb33-7d00-431c-a780-261995d86f3c', 
	sUserPassword:= '68bc2b87-a9ad-4107-814c-33cbf7ba0678', 
	eSavePositionCertificate:= eSavePositionOnPLC.ePostionHardDisk, 
	bConnected=> , 
	bError=> , 
	hrErrorCode=> , 
	eConnectionState=> , 
	eErrorMessage_Out=> );
*)

END_PROGRAM

// ---- POUs/prgWCounter_old.TcPOU
PROGRAM prgWCounter_old
VAR
	fbMBusKL6781 : FB_MBUSKL6781;
	fbmbusScan	: FB_MBUS_Scan;
	bStartScan : BOOL;
	bStopScan : BOOL;
	stComIn    AT %I*	:	ST_KL6781inData22B;
	stComOut   AT %Q*	:	ST_KL6781outData22B;
	stCom				:	ST_MBUS_Communication;
	fb_Mbus				: 	FB_MBUS_General_Water;
	sec_Address			: 	ST_MBUS_SecAdr;
	
	m_Start: BOOL;
	state: INT;
	ton_Wait: Ton;
	x: INT;							
	udint_Adress: UDINT;
	manu: INT:=1;
	int_Found: INT;							//{#lynus.ag#()}
END_VAR

CASE state OF
	0: // init
		sec_Address.usiVersion     :=0;
		state:=1;
	1: // start request
		m_Start := TRUE;
		state:=2;
	2: // wait for busy getting low
		IF fb_Mbus.bBusy = FALSE THEN		
			m_Start := FALSE;
			IF fb_Mbus.bError = TRUE THEN
				sec_Address.usiVersion := sec_Address.usiVersion+1;
				state := 3;
			ELSE
				state := 3;
				x:=x+1;
			END_IF
		END_IF
	3: // wait
		ton_Wait.IN:=TRUE;
		IF ton_Wait.Q THEN
			ton_Wait.IN:=FALSE;
			state :=1;
		END_IF
END_CASE
ton_Wait(PT:=T#500MS);


int_Found:=x;

IF sec_Address.usiVersion>251 THEN 
	sec_Address.usiVersion:=0; 
	IF manu>109 THEN 
		manu:=1;
		sec_Address.udiIdNumber:=172785;
	ELSE
		manu:=manu+1;
	END_IF
	CASE manu OF 
		1	:	sec_Address.uiManufacturer := 16#0442	;
		2	:	sec_Address.uiManufacturer := 16#0465	;
		3	:	sec_Address.uiManufacturer := 16#0467	;
		4	:	sec_Address.uiManufacturer := 16#0477	;
		5	:	sec_Address.uiManufacturer := 16#04A7	;
		6	:	sec_Address.uiManufacturer := 16#04AC	;
		7	:	sec_Address.uiManufacturer := 16#04AD	;
		8	:	sec_Address.uiManufacturer := 16#05B0	;
		9	:	sec_Address.uiManufacturer := 16#05B4	;
		10	:	sec_Address.uiManufacturer := 16#0613	;
		11	:	sec_Address.uiManufacturer := 16#08A3	;
		12	:	sec_Address.uiManufacturer := 16#08B2	;
		13	:	sec_Address.uiManufacturer := 16#0A65	;
		14	:	sec_Address.uiManufacturer := 16#0A74	;
		15	:	sec_Address.uiManufacturer := 16#0C49	;
		16	:	sec_Address.uiManufacturer := 16#0D8F	;
		17	:	sec_Address.uiManufacturer := 16#0DEE	;
		18	:	sec_Address.uiManufacturer := 16#0F4D	;
		19	:	sec_Address.uiManufacturer := 16#102E	;
		20	:	sec_Address.uiManufacturer := 16#10D3	;
		21	:	sec_Address.uiManufacturer := 16#11A5	;
		22	:	sec_Address.uiManufacturer := 16#1347	;
		23	:	sec_Address.uiManufacturer := 16#148D	;
		24	:	sec_Address.uiManufacturer := 16#14C5	;
		25	:	sec_Address.uiManufacturer := 16#1574	;
		26	:	sec_Address.uiManufacturer := 16#158D	;
		27	:	sec_Address.uiManufacturer := 16#1593	;
		28	:	sec_Address.uiManufacturer := 16#15A8	;
		29	:	sec_Address.uiManufacturer := 16#15B5	;
		30	:	sec_Address.uiManufacturer := 16#15AF	;
		31	:	sec_Address.uiManufacturer := 16#15C4	;
		32	:	sec_Address.uiManufacturer := 16#15D0	;
		33	:	sec_Address.uiManufacturer := 16#15D4	;
		34	:	sec_Address.uiManufacturer := 16#164C	;
		35	:	sec_Address.uiManufacturer := 16#166D	;
		36	:	sec_Address.uiManufacturer := 16#16B2	;
		37	:	sec_Address.uiManufacturer := 16#16F4	;
		38	:	sec_Address.uiManufacturer := 16#18A4	;
		39	:	sec_Address.uiManufacturer := 16#19AC	;
		40	:	sec_Address.uiManufacturer := 16#1C4A	;
		41	:	sec_Address.uiManufacturer := 16#1CA3	;
		42	:	sec_Address.uiManufacturer := 16#1E70	;
		43	:	sec_Address.uiManufacturer := 16#1EE6	;
		44	:	sec_Address.uiManufacturer := 16#20A7	;
		45	:	sec_Address.uiManufacturer := 16#20AC	;
		46	:	sec_Address.uiManufacturer := 16#2283	;
		47	:	sec_Address.uiManufacturer := 16#2324	;
		48	:	sec_Address.uiManufacturer := 16#246D	;
		49	:	sec_Address.uiManufacturer := 16#2485	;
		50	:	sec_Address.uiManufacturer := 16#25D6	;
		51	:	sec_Address.uiManufacturer := 16#266B	;
		52	:	sec_Address.uiManufacturer := 16#2674	;
		53	:	sec_Address.uiManufacturer := 16#2692	;
		54	:	sec_Address.uiManufacturer := 16#26EB	;
		55	:	sec_Address.uiManufacturer := 16#2C2D	;
		56	:	sec_Address.uiManufacturer := 16#2D0C	;
		57	:	sec_Address.uiManufacturer := 16#2D65	;
		58	:	sec_Address.uiManufacturer := 16#2DD8	;
		59	:	sec_Address.uiManufacturer := 16#2E4F	;
		60	:	sec_Address.uiManufacturer := 16#2E74	;
		61	:	sec_Address.uiManufacturer := 16#30AD	;
		62	:	sec_Address.uiManufacturer := 16#30E2	;
		63	:	sec_Address.uiManufacturer := 16#30E4	;
		64	:	sec_Address.uiManufacturer := 16#30FA	;
		65	:	sec_Address.uiManufacturer := 16#3101	;
		66	:	sec_Address.uiManufacturer := 16#31AC	;
		67	:	sec_Address.uiManufacturer := 16#3265	;
		68	:	sec_Address.uiManufacturer := 16#3270	;
		69	:	sec_Address.uiManufacturer := 16#32A7	;
		70	:	sec_Address.uiManufacturer := 16#327A	;
		71	:	sec_Address.uiManufacturer := 16#3424	;
		72	:	sec_Address.uiManufacturer := 16#34A9	;
		73	:	sec_Address.uiManufacturer := 16#3573	;
		74	:	sec_Address.uiManufacturer := 16#35D3	;
		75	:	sec_Address.uiManufacturer := 16#3613	;
		76	:	sec_Address.uiManufacturer := 16#3683	;
		77	:	sec_Address.uiManufacturer := 16#3933	;
		78	:	sec_Address.uiManufacturer := 16#39B3	;
		79	:	sec_Address.uiManufacturer := 16#3A4D	;
		80	:	sec_Address.uiManufacturer := 16#3DD2	;
		81	:	sec_Address.uiManufacturer := 16#4024	;
		82	:	sec_Address.uiManufacturer := 16#41A7	;
		83	:	sec_Address.uiManufacturer := 16#4249	;
		84	:	sec_Address.uiManufacturer := 16#4833	;
		85	:	sec_Address.uiManufacturer := 16#48AC	;
		86	:	sec_Address.uiManufacturer := 16#4965	;
		87	:	sec_Address.uiManufacturer := 16#4C30	;
		88	:	sec_Address.uiManufacturer := 16#4C68	;
		89	:	sec_Address.uiManufacturer := 16#4CAE	;
		90	:	sec_Address.uiManufacturer := 16#4DA3	;
		91	:	sec_Address.uiManufacturer := 16#4DA5	;
		92	:	sec_Address.uiManufacturer := 16#4DAC	;
		93	:	sec_Address.uiManufacturer := 16#4D25	;
		94	:	sec_Address.uiManufacturer := 16#4D82	;
		95	:	sec_Address.uiManufacturer := 16#4DEE	;
		96	:	sec_Address.uiManufacturer := 16#4DE6	;
		97	:	sec_Address.uiManufacturer := 16#4E0C	;
		98	:	sec_Address.uiManufacturer := 16#4E18	;
		99	:	sec_Address.uiManufacturer := 16#4ECD	;
		100	:	sec_Address.uiManufacturer := 16#5068	;
		101	:	sec_Address.uiManufacturer := 16#5130	;
		102	:	sec_Address.uiManufacturer := 16#5427	;
		103	:	sec_Address.uiManufacturer := 16#54E9	;
		104	:	sec_Address.uiManufacturer := 16#58B3	;
		105	:	sec_Address.uiManufacturer := 16#5A09	;
		106	:	sec_Address.uiManufacturer := 16#5DAF	;
		107	:	sec_Address.uiManufacturer := 16#6685	;
		108	:	sec_Address.uiManufacturer := 16#6827	;
		109	:	sec_Address.uiManufacturer := 16#6830	;
		110	:	sec_Address.uiManufacturer := 16#6936	;
	END_CASE
END_IF
		
		
fb_Mbus(	usiAddress	:= 	253,
			stSecAdr	:= 	sec_Address,
			eBaudrate   :=	E_MBUS_Baudrate.eMBus_Baud2400,
			bStart      :=	m_Start,
			stCom		:=	stCom);
	
fbMBusKL6781(
	usiRetries:= , 
	bStart:= , 
	bDisabled:= , 
	bBusy=> , 
	bReady=> , 
	bError=> , 
	eError=> , 
	stComIn:= stComIn, 
	stComOut:= stComOut, 
	stCom:= stCom);

			
(*
	
fbMBusScan(
	bStart:= , 
	bStop:= , 
	eBaudrate:= , 
	bDisabled:= , 
	bBusy=> , 
	bReady=> , 
	bError=> , 
	eError=> , 
	usiAddress=> , 
	usiCount=> , 
	arrDevice=> , 
	stCom:= stCom);
	
	*)

END_PROGRAM
